// TIA Portal project "8_Height_Sorting_Advanced" (V19)

(* hardware
DEVICE "S7-1500/ET200MP station_1"  S7-1500 station
   slot 0: "Rail_0"  Rack  6ES7 590-1***0-0AA0
   slot 1: "PLC_1"  CPU 1513-1 PN  6ES7 513-1AL02-0AB0  V2.9
      slot 3: "CPU display_1"  6ES7591-1AA00-0AA0
      slot 32768: "PROFINET interface_1"  X1
         slot 32769: "Port_1"  X1 P1
         slot 32770: "Port_2"  X1 P2
      slot 34817: "Virtual CP interface port_1"  Virtual CP interface port  Virtual CP interface port
*)

// ===== PLC "PLC_1"  CPU 1513-1 PN =====

VAR_GLOBAL   // PLC tag table "Default tag table"
   "Tag_1" AT %M0.0 : Bool;
   "Tag_2" AT %M0.6 : Bool;
   "Tag_3" AT %M0.1 : Bool;
   "Tag_4" AT %M0.7 : Bool;
   "Network 4" AT %M1.1 : Bool;
   "Network 5" AT %M1.2 : Bool;
   "Network 3" AT %M1.0 : Bool;
   "Tag_5" AT %M1.3 : Bool;
   "Tag_6" AT %M1.4 : Bool;
   "Tag_7" AT %M1.5 : Bool;
   "Network 7" AT %M1.6 : Bool;
   "Tag_8" AT %M0.2 : Bool;
   "Tag_9" AT %M1.7 : Bool;
   "Tag_10" AT %M2.5 : Bool;
   "Tag_11" AT %M2.6 : Bool;
   "Tag_12" AT %M2.0 : Bool;
   "Tag_13" AT %M2.1 : Bool;
   "Tag_14" AT %M2.2 : Bool;
   "Tag_15" AT %M2.3 : Bool;
   "Tag_16" AT %M0.3 : Bool;
   "Tag_17" AT %M0.4 : Bool;
   "Tag_18" AT %M0.5 : Bool;
   "Tag_19" AT %M2.4 : Bool;
END_VAR

VAR_GLOBAL   // PLC tag table "Tag table from XML_1"
   "Start Button" AT %I0.0 : Bool;
   "Stop Button" AT %I0.1 : Bool;
   "Palletizer box Sensor" AT %I0.2 : Bool;
   "Medium Box Sensor" AT %I0.3 : Bool;
   "Large box Sensor" AT %I0.4 : Bool;
   "At right entry" AT %I0.5 : Bool;
   "At right exit" AT %I0.6 : Bool;
   "At left entry" AT %I0.7 : Bool;
   "At left exit" AT %I1.0 : Bool;
   "At straight entry" AT %I1.1 : Bool;
   "At straight exit" AT %I1.2 : Bool;
   "At back" AT %I1.3 : Bool;
   "At front" AT %I1.4 : Bool;
   "At load position" AT %I1.5 : Bool;
   "At unload position" AT %I1.6 : Bool;
   "Start Button (LED)" AT %Q0.0 : Bool;
   "Stop Button (LED)" AT %Q0.1 : Bool;
   "Entry conveyor" AT %Q0.2 : Bool;
   "Right conveyor" AT %Q0.3 : Bool;
   "Left conveyor" AT %Q0.4 : Bool;
   "Straight Conveyor" AT %Q0.5 : Bool;
   "Load" AT %Q0.6 : Bool;
   "Unload" AT %Q0.7 : Bool;
   "Turn" AT %Q1.0 : Bool;
   "Green indicator" AT %Q1.1 : Bool;
   "Red indicator" AT %Q1.2 : Bool;
   "Pallet Box Count" AT %QD30 : DInt;
   "Medium Box Count" AT %QD34 : DInt;
   "Large Box Count" AT %QD38 : DInt;
END_VAR

// folder: System blocks/Program resources

DATA_BLOCK "IEC_Counter_0_DB"   // DB1
{ S7_Optimized_Access := 'TRUE' }
AUTHOR : Simatic
FAMILY : IEC
NAME : CNTR
VERSION : 1.0
// stored: InstanceOfName IEC_COUNTER
"IEC_COUNTER"
BEGIN
END_DATA_BLOCK

DATA_BLOCK "IEC_Counter_0_DB_1"   // DB2
{ S7_Optimized_Access := 'TRUE' }
AUTHOR : Simatic
FAMILY : IEC
NAME : CNTR
VERSION : 1.0
// stored: InstanceOfName IEC_COUNTER
"IEC_COUNTER"
BEGIN
END_DATA_BLOCK

DATA_BLOCK "IEC_Counter_0_DB_2"   // DB3
{ S7_Optimized_Access := 'TRUE' }
AUTHOR : Simatic
FAMILY : IEC
NAME : CNTR
VERSION : 1.0
// stored: InstanceOfName IEC_COUNTER
"IEC_COUNTER"
BEGIN
END_DATA_BLOCK

// folder: (top level)

ORGANIZATION_BLOCK "Main"   // OB1, LAD, ProgramCycle
TITLE = "Main Program Sweep (Cycle)"
{ S7_Optimized_Access := 'TRUE' }
VERSION : 0.1
   VAR_INPUT
      Initial_Call : Bool;   // Initial call of this OB
      Remanence : Bool;   // =True, if remanent data are available
   END_VAR
   VAR_TEMP   // added for the SCL form of the ladder/FBD networks
      _w1 : Bool;
      _w2 : Bool;
      _w3 : Bool;
   END_VAR
BEGIN

REGION Network 1: Intitialize LED and Indicator
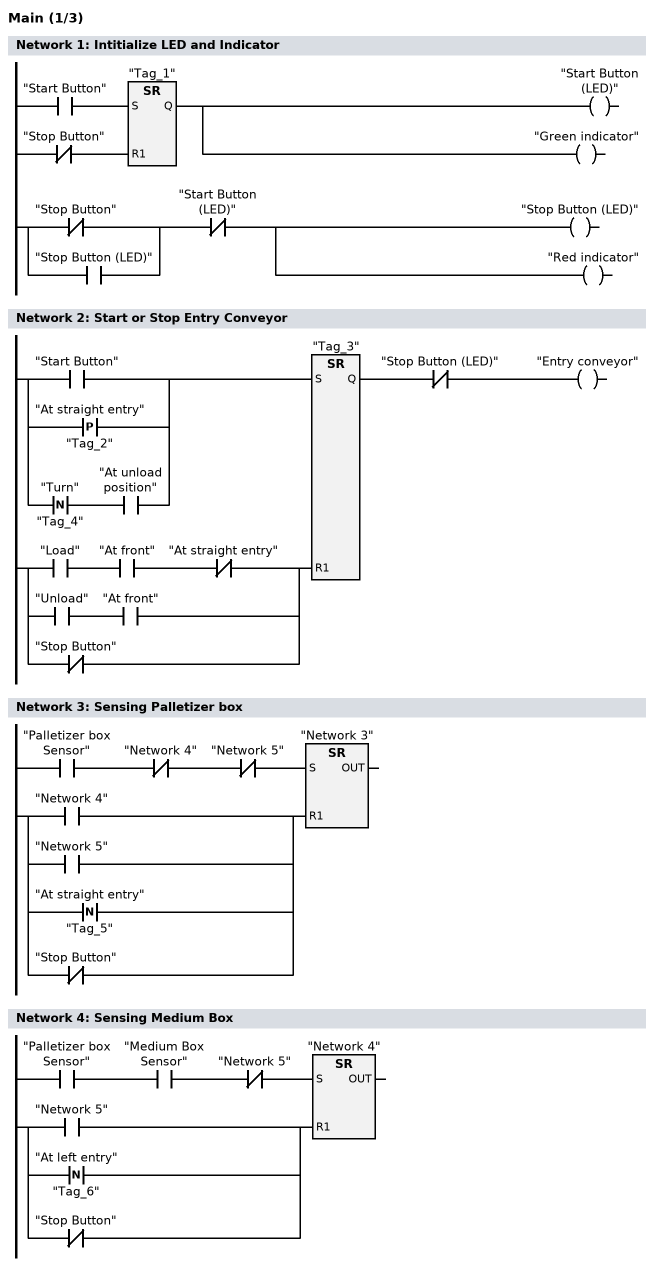
   RUNG wire#powerrail
      Contact( "Start Button" )
      S_SR(operand := "Tag_1", r1 := wire#w1)
      wire#w2
      Coil( "Start Button (LED)" )
   END_RUNG
   RUNG wire#powerrail
      I_Contact( "Stop Button" )
   END_RUNG wire#w1
   RUNG wire#w2
      Coil( "Green indicator" )
   END_RUNG
   RUNG wire#powerrail
      I_Contact( "Stop Button" )
      wire#w3
      I_Contact( "Start Button (LED)" )
      wire#w4
      Coil( "Stop Button (LED)" )
   END_RUNG
   RUNG wire#powerrail
      Contact( "Stop Button (LED)" )
   END_RUNG wire#w3
   RUNG wire#w4
      Coil( "Red indicator" )
   END_RUNG
   // the same network as SCL:
   IF "Start Button" THEN
       "Tag_1" := TRUE;   // SR flip-flop
   END_IF;
   IF NOT "Stop Button" THEN "Tag_1" := FALSE; END_IF;
   "Start Button (LED)" := "Tag_1";
   "Green indicator" := "Tag_1";
   "Stop Button (LED)" := (NOT "Stop Button" OR "Stop Button (LED)") AND NOT "Start Button (LED)";
   "Red indicator" := "Stop Button (LED)";
END_REGION

REGION Network 2: Start or Stop Entry Conveyor
   RUNG wire#powerrail
      Contact( "Start Button" )
      wire#w1
      S_SR(operand := "Tag_3", r1 := wire#w2)
      I_Contact( "Stop Button (LED)" )
      Coil( "Entry conveyor" )
   END_RUNG
   RUNG wire#powerrail
      P_Contact(operand := "At straight entry", bit := "Tag_2")
   END_RUNG wire#w1
   RUNG wire#powerrail
      N_Contact(operand := "Turn", bit := "Tag_4")
      Contact( "At unload position" )
   END_RUNG wire#w1
   RUNG wire#powerrail
      Contact( "Load" )
      Contact( "At front" )
      I_Contact( "At straight entry" )
   END_RUNG wire#w2
   RUNG wire#powerrail
      Contact( "Unload" )
      Contact( "At front" )
   END_RUNG wire#w2
   RUNG wire#powerrail
      I_Contact( "Stop Button" )
   END_RUNG wire#w2
   // the same network as SCL:
   #_w1 := "At straight entry" AND NOT "Tag_2";   // rising edge of "At straight entry"
   "Tag_2" := "At straight entry";
   #_w2 := NOT "Turn" AND "Tag_4";   // falling edge of "Turn"
   "Tag_4" := "Turn";
   IF "Start Button" OR #_w1 OR (#_w2 AND "At unload position") THEN
       "Tag_3" := TRUE;   // SR flip-flop
   END_IF;
   IF ("Load" AND "At front" AND NOT "At straight entry") OR ("Unload" AND "At front") OR NOT "Stop Button" THEN
       "Tag_3" := FALSE;
   END_IF;
   "Entry conveyor" := "Tag_3" AND NOT "Stop Button (LED)";
END_REGION

REGION Network 3: Sensing Palletizer box
   RUNG wire#powerrail
      Contact( "Palletizer box Sensor" )
      I_Contact( "Network 4" )
      I_Contact( "Network 5" )
      S_SR(operand := "Network 3", r1 := wire#w1)
   END_RUNG
   RUNG wire#powerrail
      Contact( "Network 4" )
   END_RUNG wire#w1
   RUNG wire#powerrail
      Contact( "Network 5" )
   END_RUNG wire#w1
   RUNG wire#powerrail
      N_Contact(operand := "At straight entry", bit := "Tag_5")
   END_RUNG wire#w1
   RUNG wire#powerrail
      I_Contact( "Stop Button" )
   END_RUNG wire#w1
   // the same network as SCL:
   #_w1 := NOT "At straight entry" AND "Tag_5";   // falling edge of "At straight entry"
   "Tag_5" := "At straight entry";
   IF "Palletizer box Sensor" AND NOT "Network 4" AND NOT "Network 5" THEN
       "Network 3" := TRUE;   // SR flip-flop
   END_IF;
   IF "Network 4" OR "Network 5" OR #_w1 OR NOT "Stop Button" THEN "Network 3" := FALSE; END_IF;
END_REGION

REGION Network 4: Sensing Medium Box
   RUNG wire#powerrail
      Contact( "Palletizer box Sensor" )
      Contact( "Medium Box Sensor" )
      I_Contact( "Network 5" )
      S_SR(operand := "Network 4", r1 := wire#w1)
   END_RUNG
   RUNG wire#powerrail
      Contact( "Network 5" )
   END_RUNG wire#w1
   RUNG wire#powerrail
      N_Contact(operand := "At left entry", bit := "Tag_6")
   END_RUNG wire#w1
   RUNG wire#powerrail
      I_Contact( "Stop Button" )
   END_RUNG wire#w1
   // the same network as SCL:
   #_w1 := NOT "At left entry" AND "Tag_6";   // falling edge of "At left entry"
   "Tag_6" := "At left entry";
   IF "Palletizer box Sensor" AND "Medium Box Sensor" AND NOT "Network 5" THEN
       "Network 4" := TRUE;   // SR flip-flop
   END_IF;
   IF "Network 5" OR #_w1 OR NOT "Stop Button" THEN "Network 4" := FALSE; END_IF;
END_REGION

REGION Network 5: Sensing Large Box
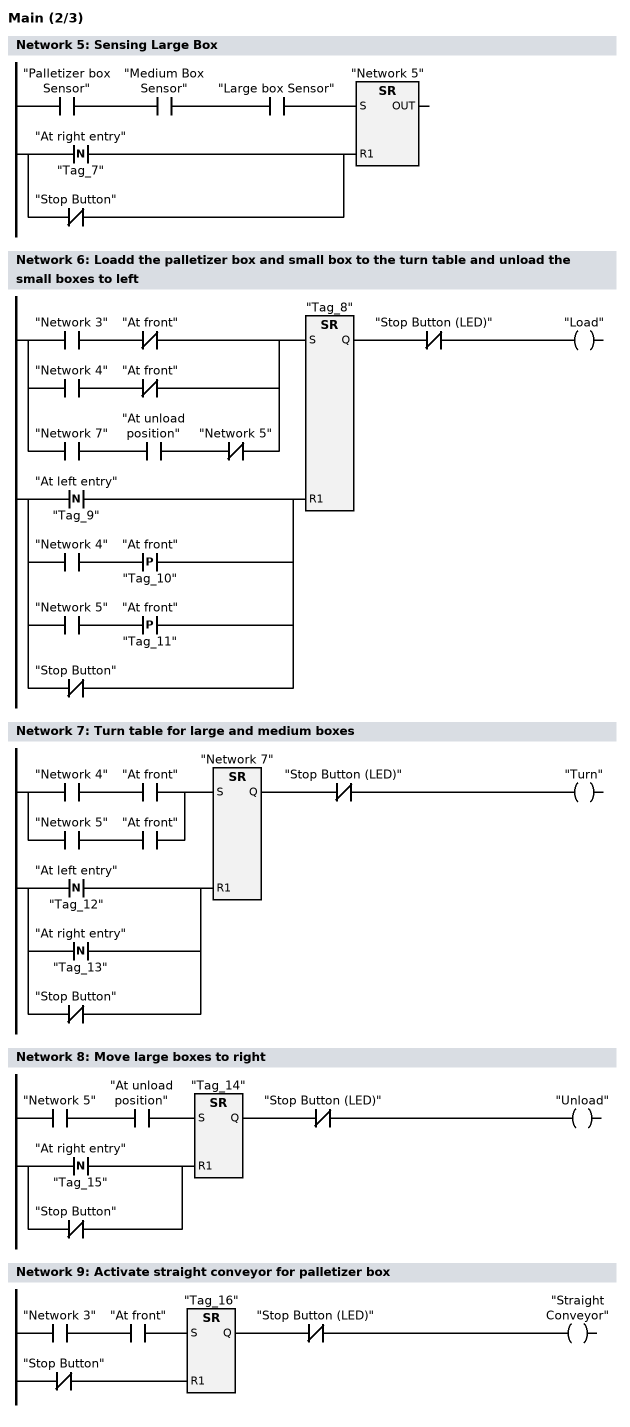
   RUNG wire#powerrail
      Contact( "Palletizer box Sensor" )
      Contact( "Medium Box Sensor" )
      Contact( "Large box Sensor" )
      S_SR(operand := "Network 5", r1 := wire#w1)
   END_RUNG
   RUNG wire#powerrail
      N_Contact(operand := "At right entry", bit := "Tag_7")
   END_RUNG wire#w1
   RUNG wire#powerrail
      I_Contact( "Stop Button" )
   END_RUNG wire#w1
   // the same network as SCL:
   #_w1 := NOT "At right entry" AND "Tag_7";   // falling edge of "At right entry"
   "Tag_7" := "At right entry";
   IF "Palletizer box Sensor" AND "Medium Box Sensor" AND "Large box Sensor" THEN
       "Network 5" := TRUE;   // SR flip-flop
   END_IF;
   IF #_w1 OR NOT "Stop Button" THEN "Network 5" := FALSE; END_IF;
END_REGION

REGION Network 6: Loadd the palletizer box and small box to the turn table and unload the small boxes to left
   RUNG wire#powerrail
      Contact( "Network 3" )
      I_Contact( "At front" )
      wire#w1
      S_SR(operand := "Tag_8", r1 := wire#w2)
      I_Contact( "Stop Button (LED)" )
      Coil( "Load" )
   END_RUNG
   RUNG wire#powerrail
      Contact( "Network 4" )
      I_Contact( "At front" )
   END_RUNG wire#w1
   RUNG wire#powerrail
      Contact( "Network 7" )
      Contact( "At unload position" )
      I_Contact( "Network 5" )
   END_RUNG wire#w1
   RUNG wire#powerrail
      N_Contact(operand := "At left entry", bit := "Tag_9")
   END_RUNG wire#w2
   RUNG wire#powerrail
      Contact( "Network 4" )
      P_Contact(operand := "At front", bit := "Tag_10")
   END_RUNG wire#w2
   RUNG wire#powerrail
      Contact( "Network 5" )
      P_Contact(operand := "At front", bit := "Tag_11")
   END_RUNG wire#w2
   RUNG wire#powerrail
      I_Contact( "Stop Button" )
   END_RUNG wire#w2
   // the same network as SCL:
   #_w1 := NOT "At left entry" AND "Tag_9";   // falling edge of "At left entry"
   "Tag_9" := "At left entry";
   #_w2 := "Network 4" AND "At front" AND NOT "Tag_10";   // rising edge of "At front"
   "Tag_10" := "At front";
   #_w3 := "Network 5" AND "At front" AND NOT "Tag_11";   // rising edge of "At front"
   "Tag_11" := "At front";
   IF ("Network 3" AND NOT "At front") OR ("Network 4" AND NOT "At front") OR ("Network 7" AND "At unload position" AND NOT "Network 5") THEN
       "Tag_8" := TRUE;   // SR flip-flop
   END_IF;
   IF #_w1 OR #_w2 OR #_w3 OR NOT "Stop Button" THEN "Tag_8" := FALSE; END_IF;
   "Load" := "Tag_8" AND NOT "Stop Button (LED)";
END_REGION

REGION Network 7: Turn table for large and medium boxes
   RUNG wire#powerrail
      Contact( "Network 4" )
      Contact( "At front" )
      wire#w1
      S_SR(operand := "Network 7", r1 := wire#w2)
      I_Contact( "Stop Button (LED)" )
      Coil( "Turn" )
   END_RUNG
   RUNG wire#powerrail
      Contact( "Network 5" )
      Contact( "At front" )
   END_RUNG wire#w1
   RUNG wire#powerrail
      N_Contact(operand := "At left entry", bit := "Tag_12")
   END_RUNG wire#w2
   RUNG wire#powerrail
      N_Contact(operand := "At right entry", bit := "Tag_13")
   END_RUNG wire#w2
   RUNG wire#powerrail
      I_Contact( "Stop Button" )
   END_RUNG wire#w2
   // the same network as SCL:
   #_w1 := NOT "At left entry" AND "Tag_12";   // falling edge of "At left entry"
   "Tag_12" := "At left entry";
   #_w2 := NOT "At right entry" AND "Tag_13";   // falling edge of "At right entry"
   "Tag_13" := "At right entry";
   IF ("Network 4" AND "At front") OR ("Network 5" AND "At front") THEN
       "Network 7" := TRUE;   // SR flip-flop
   END_IF;
   IF #_w1 OR #_w2 OR NOT "Stop Button" THEN "Network 7" := FALSE; END_IF;
   "Turn" := "Network 7" AND NOT "Stop Button (LED)";
END_REGION

REGION Network 8: Move large boxes to right
   RUNG wire#powerrail
      Contact( "Network 5" )
      Contact( "At unload position" )
      S_SR(operand := "Tag_14", r1 := wire#w1)
      I_Contact( "Stop Button (LED)" )
      Coil( "Unload" )
   END_RUNG
   RUNG wire#powerrail
      N_Contact(operand := "At right entry", bit := "Tag_15")
   END_RUNG wire#w1
   RUNG wire#powerrail
      I_Contact( "Stop Button" )
   END_RUNG wire#w1
   // the same network as SCL:
   #_w1 := NOT "At right entry" AND "Tag_15";   // falling edge of "At right entry"
   "Tag_15" := "At right entry";
   IF "Network 5" AND "At unload position" THEN
       "Tag_14" := TRUE;   // SR flip-flop
   END_IF;
   IF #_w1 OR NOT "Stop Button" THEN "Tag_14" := FALSE; END_IF;
   "Unload" := "Tag_14" AND NOT "Stop Button (LED)";
END_REGION

REGION Network 9: Activate straight conveyor for palletizer box
   RUNG wire#powerrail
      Contact( "Network 3" )
      Contact( "At front" )
      S_SR(operand := "Tag_16", r1 := wire#w1)
      I_Contact( "Stop Button (LED)" )
      Coil( "Straight Conveyor" )
   END_RUNG
   RUNG wire#powerrail
      I_Contact( "Stop Button" )
   END_RUNG wire#w1
   // the same network as SCL:
   IF "Network 3" AND "At front" THEN
       "Tag_16" := TRUE;   // SR flip-flop
   END_IF;
   IF NOT "Stop Button" THEN "Tag_16" := FALSE; END_IF;
   "Straight Conveyor" := "Tag_16" AND NOT "Stop Button (LED)";
END_REGION

REGION Network 10: Activate right conveyor for large box
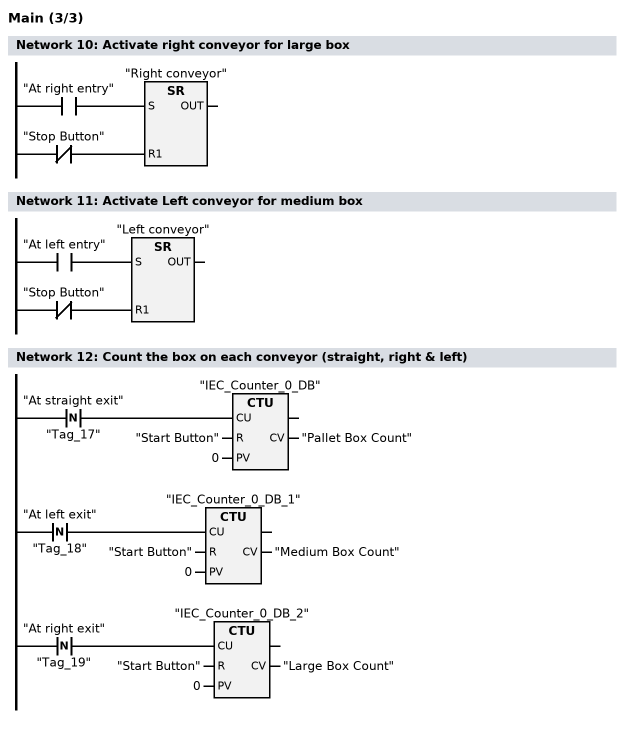
   RUNG wire#powerrail
      Contact( "At right entry" )
      S_SR(operand := "Right conveyor", r1 := wire#w1)
   END_RUNG
   RUNG wire#powerrail
      I_Contact( "Stop Button" )
   END_RUNG wire#w1
   // the same network as SCL:
   IF "At right entry" THEN
       "Right conveyor" := TRUE;   // SR flip-flop
   END_IF;
   IF NOT "Stop Button" THEN "Right conveyor" := FALSE; END_IF;
END_REGION

REGION Network 11: Activate Left conveyor for medium box
   RUNG wire#powerrail
      Contact( "At left entry" )
      S_SR(operand := "Left conveyor", r1 := wire#w1)
   END_RUNG
   RUNG wire#powerrail
      I_Contact( "Stop Button" )
   END_RUNG wire#w1
   // the same network as SCL:
   IF "At left entry" THEN
       "Left conveyor" := TRUE;   // SR flip-flop
   END_IF;
   IF NOT "Stop Button" THEN "Left conveyor" := FALSE; END_IF;
END_REGION

REGION Network 12: Count the box on each conveyor (straight, right & left)
   #_w1 := NOT "At straight exit" AND "Tag_17";   // falling edge of "At straight exit"
   "Tag_17" := "At straight exit";
   "IEC_Counter_0_DB".CTU(CU := #_w1, R := "Start Button", PV := 0, CV => "Pallet Box Count");
   #_w2 := NOT "At left exit" AND "Tag_18";   // falling edge of "At left exit"
   "Tag_18" := "At left exit";
   "IEC_Counter_0_DB_1".CTU(CU := #_w2, R := "Start Button", PV := 0, CV => "Medium Box Count");
   #_w3 := NOT "At right exit" AND "Tag_19";   // falling edge of "At right exit"
   "Tag_19" := "At right exit";
   "IEC_Counter_0_DB_2".CTU(CU := #_w3, R := "Start Button", PV := 0, CV => "Large Box Count");
END_REGION
END_ORGANIZATION_BLOCK